// TIA Portal V20 export
TYPE "LER_typeZoneOperationEnable"
// stored: Access Published
   STRUCT
      DoorLockEnable : Bool;
      DoorUnLockEnable : Bool;
      OpHMIenable : Bool;
      PHMIenable : Bool;
   END_STRUCT;
END_TYPE
